(* IEC 61131-3 sources: cc_kush_rewrite/POUs/Dumper/POU/Hardware, 4 files *)

(* ---- FB_DumperConveyorMotors.st ---- *)
FUNCTION_BLOCK FB_DumperConveyorMotors
VAR_INPUT
	Dumper : REFERENCE TO ST_Dumper;
	xStart : BOOL;              // Команда запуска
	xStop : BOOL;               // Команда остановки
	xEmergencyStop : BOOL;      // Аварийная остановка (импульсная)
	xReset : BOOL;              // Сброс аварии (импульсная)
	rTargetFrequency : REAL;    // Целевая частота моторов
END_VAR
VAR_OUTPUT
	eStage : E_StageActuator;   // Текущая стадия
	rCurrentFrequency : REAL;   // Текущая частота моторов (среднее значение)
	xStartingTimeout : BOOL;    // Флаг тайм-аута запуска (STARTING слишком долго)
	xStoppingTimeout : BOOL;    // Флаг тайм-аута остановки (STOPPING слишком долго)
	xVFD_FeedbackLostTimeout : BOOL; // Флаг: потеря обратной связи VFD во время работы (не восстановилась за TIME_TIMEOUT_VFD_FEEDBACK_LOST)
END_VAR
VAR
	STAGE : E_StageActuator := E_StageActuator.IDLE;

	// Подстадии запуска
	nStartingSubstage : INT := 0;
	// 0 - RELEASE_BRAKE: Отпускание тормоза
	// 1 - WAIT_BRAKE_FEEDBACK: Ожидание обратной связи тормоза
	// 2 - START_VFD: Запуск VFD

	// Подстадии остановки
	nStoppingSubstage : INT := 0;
	// 0 - Нормальная работа
	// 1 - STOP_VFD: Остановка VFD
	// 2 - WAIT_VFD_STOP: Ожидание остановки VFD
	// 3 - ACTIVATE_BRAKE: Активация тормоза
	// 4 - WAIT_BRAKE_FEEDBACK: Ожидание обратной связи тормоза

	// Таймер задержки включения тормоза
	tonTimerEnableBrake : TON;

	// Таймер контроля времени запуска (STARTING → WORK)
	tonTimerStarting : TON;

	// Таймер контроля времени остановки (STOPPING → IDLE)
	tonTimerStopping : TON;

	// Таймер контроля потери обратной связи VFD во время работы
	tonTimerVFD_FeedbackLost : TON;

	// Флаг запуска таймера (защита от зацикливания)
	xBrakeTimerStarted : BOOL := FALSE;
END_VAR

// ========================================
// FB_DumperConveyorMotors - Управление моторами конвейера отвалообразователя
// ========================================
//
// НАЗНАЧЕНИЕ:
// - Управление двумя моторами конвейера (22 кВт каждый)
// - Прямой пуск (без плавного разгона)
// - Последовательная остановка (VFD → тормоз)
// - Не знает про ППЗ и верхнеуровневую логику
// - Просто выполняет команды START/STOP
//
// ВХОДЫ:
// - xStart: команда запуска моторов
// - xStop: команда остановки моторов
// - xEmergencyStop: аварийная остановка (импульсная)
// - xReset: сброс аварии (импульсная)
// - rTargetFrequency: целевая частота (Гц)
//
// ВЫХОДЫ:
// - eStage: текущая стадия (IDLE/STARTING/WORK/STOPPING/FAULT)
// - rCurrentFrequency: текущая частота моторов
//
// ========================================

// ========================================
// ПРИОРИТЕТНАЯ ОБРАБОТКА АВАРИЙНОЙ ОСТАНОВКИ
// ========================================

IF xEmergencyStop THEN
	// Аварийная остановка: немедленное выключение VFD
	Dumper.MotorConveyor[1].VFD.qxStart := FALSE;
	Dumper.MotorConveyor[2].VFD.qxStart := FALSE;

	// Активация тормоза
	Dumper.qxBreakerConveyor := FALSE;

	// Переход в FAULT
	STAGE := E_StageActuator.FAULT;
	nStartingSubstage := 0;
	nStoppingSubstage := 0;
	tonTimerEnableBrake(IN := FALSE);
	tonTimerStarting(IN := FALSE);
	tonTimerStopping(IN := FALSE);
	xBrakeTimerStarted := FALSE;
END_IF

// Тайм-аут запуска: если слишком долго в STARTING → аварийная остановка
tonTimerStarting(
	IN := (STAGE = E_StageActuator.STARTING),
	PT := TIME_TIMEOUT_START_DUMPER_CONVEYOR
);

IF tonTimerStarting.Q THEN
	xStartingTimeout := TRUE;
	// Аварийная остановка: немедленное выключение VFD
	Dumper.MotorConveyor[1].VFD.qxStart := FALSE;
	Dumper.MotorConveyor[2].VFD.qxStart := FALSE;
	// Активация тормоза
	Dumper.qxBreakerConveyor := FALSE;
	// Переход в FAULT
	STAGE := E_StageActuator.FAULT;
	nStartingSubstage := 0;
	tonTimerStarting(IN := FALSE);
END_IF

// Тайм-аут остановки: если слишком долго в STOPPING → аварийная остановка
tonTimerStopping(
	IN := (STAGE = E_StageActuator.STOPPING),
	PT := TIME_TIMEOUT_STOP_DUMPER_CONVEYOR
);

IF tonTimerStopping.Q THEN
	xStoppingTimeout := TRUE;
	// Аварийная остановка: немедленное выключение VFD
	Dumper.MotorConveyor[1].VFD.qxStart := FALSE;
	Dumper.MotorConveyor[2].VFD.qxStart := FALSE;
	// Активация тормоза
	Dumper.qxBreakerConveyor := FALSE;
	// Переход в FAULT
	STAGE := E_StageActuator.FAULT;
	nStoppingSubstage := 0;
	tonTimerStopping(IN := FALSE);
END_IF

// Контроль потери обратной связи VFD во время работы
// Если VFD был в работе (WORK) и обратная связь пропала - включаем таймер
// Если обратная связь не вернулась в течение TIME_TIMEOUT_VFD_FEEDBACK_LOST → аварийная остановка
tonTimerVFD_FeedbackLost(
	IN := (STAGE = E_StageActuator.WORK) AND
	      (NOT Dumper.MotorConveyor[1].VFD.fbStateIsWorking.qxSignal
	       OR NOT Dumper.MotorConveyor[2].VFD.fbStateIsWorking.qxSignal),
	PT := TIME_TIMEOUT_VFD_FEEDBACK_LOST
);

IF tonTimerVFD_FeedbackLost.Q THEN
	xVFD_FeedbackLostTimeout := TRUE;
	// Аварийная остановка: немедленное выключение VFD
	Dumper.MotorConveyor[1].VFD.qxStart := FALSE;
	Dumper.MotorConveyor[2].VFD.qxStart := FALSE;
	// Активация тормоза
	Dumper.qxBreakerConveyor := FALSE;
	// Переход в FAULT
	STAGE := E_StageActuator.FAULT;
	tonTimerVFD_FeedbackLost(IN := FALSE);
END_IF

// ========================================
// АВТОМАТ УПРАВЛЕНИЯ МОТОРАМИ
// ========================================

CASE STAGE OF
	E_StageActuator.IDLE:
		// Сброс подстадий
		nStartingSubstage := 0;
		nStoppingSubstage := 0;

		// Сброс флага таймера тормоза
		xBrakeTimerStarted := FALSE;

		// Тормоз активен (удерживает механизм)
		Dumper.qxBreakerConveyor := FALSE;

		// Команда запуска
		IF xStart AND NOT xEmergencyStop THEN
			STAGE := E_StageActuator.STARTING;
		END_IF

	E_StageActuator.STARTING:
		// Проверка команды остановки во время запуска
		IF xStop THEN
			// Прервать запуск и перейти к остановке
			STAGE := E_StageActuator.STOPPING;
			nStartingSubstage := 0;
			nStoppingSubstage := 1; // Начать процедуру остановки
		END_IF

		// Последовательный запуск: Тормоз → VFD → Разгон
		CASE nStartingSubstage OF
			0: // RELEASE_BRAKE - Отпускание тормоза
				// Отпустить тормоз (1 = тормоз отпущен)
				Dumper.qxBreakerConveyor := TRUE;

				// Переход к следующей подстадии
				nStartingSubstage := 1;

			1: // WAIT_BRAKE_FEEDBACK - Ожидание обратной связи тормоза
				// Получить обратную связь реле тормоза
				IF Dumper.fbBreakerConveyor.qxSignal THEN
					// Обратная связь получена, переходим к запуску VFD
					nStartingSubstage := 2;
				END_IF

			2: // START_VFD - Запуск VFD
				// Команда ПУСК на частотный преобразователь
				Dumper.MotorConveyor[1].VFD.qxStart := TRUE;
				Dumper.MotorConveyor[2].VFD.qxStart := TRUE;

				// Если оба VFD запущены (обратная связь)
				IF Dumper.MotorConveyor[1].VFD.fbStateIsWorking.qxSignal
					AND Dumper.MotorConveyor[2].VFD.fbStateIsWorking.qxSignal
				THEN
					// Переход в режим WORK
					STAGE := E_StageActuator.WORK;
					nStartingSubstage := 0;
				END_IF
		END_CASE;

	E_StageActuator.WORK:
		// Нормальная работа
		// Команда остановки - переход в STOPPING
		IF xStop THEN
			STAGE := E_StageActuator.STOPPING;
			nStoppingSubstage := 0;
		END_IF

	E_StageActuator.STOPPING:
		// Штатная остановка через подстадии
		CASE nStoppingSubstage OF
			0: // STOP_VFD - Остановка VFD
				// Отключить команду пуска на VFD
				Dumper.MotorConveyor[1].VFD.qxStart := FALSE;
				Dumper.MotorConveyor[2].VFD.qxStart := FALSE;

				nStoppingSubstage := 1;

			1: // WAIT_VFD_STOP - Ожидание остановки VFD
				// Проверить обратную связь VFD о выключении
				IF NOT Dumper.MotorConveyor[1].VFD.fbStateIsWorking.qxSignal
					AND NOT Dumper.MotorConveyor[2].VFD.fbStateIsWorking.qxSignal
				THEN
					nStoppingSubstage := 2;
				END_IF

			2: // ACTIVATE_BRAKE - Активация тормоза с задержкой
				// Включение таймера на задержку тормоза (один раз)
				IF NOT xBrakeTimerStarted THEN
					xBrakeTimerStarted := TRUE;
				END_IF

				tonTimerEnableBrake(IN := xBrakeTimerStarted, PT := T#5S);

				IF tonTimerEnableBrake.Q THEN
					// Снять сигнал с тормоза (FALSE = активен)
					Dumper.qxBreakerConveyor := FALSE;
					tonTimerEnableBrake(IN := FALSE);
					xBrakeTimerStarted := FALSE;
					nStoppingSubstage := 3;
				END_IF

			3: // Переход в IDLE
				STAGE := E_StageActuator.IDLE;
				nStoppingSubstage := 0;
		END_CASE;

	E_StageActuator.FAULT:
		// Состояние аварии - ожидание сброса
		// Выход из FAULT по команде xReset
		IF xReset THEN
			STAGE := E_StageActuator.IDLE;
			xStartingTimeout := FALSE; // Сброс флага тайм-аута запуска
			xStoppingTimeout := FALSE; // Сброс флага тайм-аута остановки
			xVFD_FeedbackLostTimeout := FALSE; // Сброс флага потери обратной связи VFD
		END_IF
END_CASE;

// ========================================
// ЗАДАНИЕ ЧАСТОТЫ МОТОРОВ
// ========================================

// Установка частоты напрямую в аналоговый выход VFD
// В режимах STARTING и WORK частота = rTargetFrequency (VFD должен знать целевую частоту до запуска)
// В остальных режимах (IDLE, STOPPING, FAULT) частота = 0
IF STAGE = E_StageActuator.STARTING OR STAGE = E_StageActuator.WORK THEN
	Dumper.MotorConveyor[1].VFD.qrOutFrequency := rTargetFrequency;
	Dumper.MotorConveyor[2].VFD.qrOutFrequency := rTargetFrequency;
ELSE
	Dumper.MotorConveyor[1].VFD.qrOutFrequency := 0.0;
	Dumper.MotorConveyor[2].VFD.qrOutFrequency := 0.0;
END_IF;

// ========================================
// ВЫХОДЫ
// ========================================

// Текущая стадия
eStage := STAGE;

// Текущая частота (среднее значение двух моторов)
rCurrentFrequency := (Dumper.MotorConveyor[1].VFD.rActualFrequency
                    + Dumper.MotorConveyor[2].VFD.rActualFrequency) / 2.0;

END_FUNCTION_BLOCK

(* ---- FB_DumperMotorErrors.st ---- *)
FUNCTION_BLOCK FB_DumperMotorErrors
VAR_INPUT
	Dumper : REFERENCE TO ST_Dumper;
	xReset : BOOL; // Команда сброса зафиксированных ошибок
END_VAR
VAR_OUTPUT
	// Ошибки моторов конвейера
	xErrorMotorConv1 : BOOL;
	xErrorMotorConv2 : BOOL;
	xErrorMotorConv_Any : BOOL;

	// Ошибки моторов поворота
	xErrorMotorRot1 : BOOL;
	xErrorMotorRot2 : BOOL;
	xErrorMotorRot_Any : BOOL;

	// Агрегированный выход ошибок
	xErrorMotors : BOOL; // Любая ошибка моторов (VFD failure)

	// Готовность VFD (дискретный сигнал "Готов к пуску")
	xVFD_ReadyConv1 : BOOL; // VFD мотора конвейера 1 готов
	xVFD_ReadyConv2 : BOOL; // VFD мотора конвейера 2 готов
	xVFD_ReadyConv_All : BOOL; // Все VFD конвейера готовы

	xVFD_ReadyRot1 : BOOL; // VFD мотора поворота 1 готов
	xVFD_ReadyRot2 : BOOL; // VFD мотора поворота 2 готов
	xVFD_ReadyRot_All : BOOL; // Все VFD поворота готовы

	xVFD_Ready_All : BOOL; // Все VFD готовы к пуску

	// Состояние автоматических выключателей (QF)
	// TRUE = включен, FALSE = выключен
	// Не является ошибкой, но влияет на готовность к запуску
	xQF_OkConv1 : BOOL; // QF мотора конвейера 1 включен
	xQF_OkConv2 : BOOL; // QF мотора конвейера 2 включен
	xQF_OkConv_All : BOOL; // Все QF конвейера включены

	xQF_OkRot1 : BOOL; // QF мотора поворота 1 включен
	xQF_OkRot2 : BOOL; // QF мотора поворота 2 включен
	xQF_OkRot_All : BOOL; // Все QF поворота включены

	xQF_Ok_All : BOOL; // Все QF включены
END_VAR
VAR
	// Внутренние переменные для текущих состояний ошибок (без фиксации)
	_xCurrentErrorMotorConv1 : BOOL;
	_xCurrentErrorMotorConv2 : BOOL;
	_xCurrentErrorMotorRot1 : BOOL;
	_xCurrentErrorMotorRot2 : BOOL;

	// RS-триггеры для фиксации ошибок
	_fbLatchErrorMotorConv1 : RS;
	_fbLatchErrorMotorConv2 : RS;
	_fbLatchErrorMotorRot1 : RS;
	_fbLatchErrorMotorRot2 : RS;
END_VAR

// ========================================
// FB_DumperMotorErrors - Проверка ошибок моторов отвалообразователя
// ========================================
//
// НАЗНАЧЕНИЕ:
// - Проверка всех моторов отвалообразователя на ошибки
// - Фиксация ошибок через RS-триггеры (память до сброса)
// - Формирование индивидуальных флагов ошибок
// - Агрегирование ошибок
//
// МОТОРЫ:
// - MotorConveyor[1..2]: Моторы конвейера (22 кВт)
// - MotorRotation[1..2]: Моторы поворота (3 кВт)
//
// ПРОВЕРЯЕМЫЕ ОШИБКИ:
// - Ошибка VFD (fbStateFailure: 0 = ошибка, 1 = норма, NC контакт)
//
// ПРОВЕРЯЕМАЯ ГОТОВНОСТЬ:
// - Готовность VFD (fbStateRdyToStart: 1 = готов, 0 = не готов, NO контакт)
//
// ЛОГИКА ФИКСАЦИИ:
// - При возникновении ошибки она фиксируется (SET в RS-триггер)
// - Ошибка сохраняется даже после устранения неисправности
// - Сброс всех зафиксированных ошибок через вход xReset
//
// ========================================

// ========================================
// ПРОВЕРКА МОТОРОВ КОНВЕЙЕРА
// ========================================

// Мотор конвейера 1
// fbStateFailure - NC контакт: 0 = ошибка VFD, 1 = норма
_xCurrentErrorMotorConv1 := NOT Dumper.MotorConveyor[1].VFD.fbStateFailure.qxSignal;

// Мотор конвейера 2
_xCurrentErrorMotorConv2 := NOT Dumper.MotorConveyor[2].VFD.fbStateFailure.qxSignal;

// Фиксируем ошибки через RS-триггеры (SET при ошибке, RESET по команде xReset)
_fbLatchErrorMotorConv1(SET := _xCurrentErrorMotorConv1, RESET1 := xReset);
_fbLatchErrorMotorConv2(SET := _xCurrentErrorMotorConv2, RESET1 := xReset);

// Выходы - зафиксированные ошибки
xErrorMotorConv1 := _fbLatchErrorMotorConv1.Q1;
xErrorMotorConv2 := _fbLatchErrorMotorConv2.Q1;

xErrorMotorConv_Any := xErrorMotorConv1 OR xErrorMotorConv2;

// ========================================
// ПРОВЕРКА МОТОРОВ ПОВОРОТА
// ========================================

// Мотор поворота 1
_xCurrentErrorMotorRot1 := NOT Dumper.MotorRotation[1].VFD.fbStateFailure.qxSignal;

// Мотор поворота 2
_xCurrentErrorMotorRot2 := NOT Dumper.MotorRotation[2].VFD.fbStateFailure.qxSignal;

// Фиксируем ошибки через RS-триггеры (SET при ошибке, RESET по команде xReset)
_fbLatchErrorMotorRot1(SET := _xCurrentErrorMotorRot1, RESET1 := xReset);
_fbLatchErrorMotorRot2(SET := _xCurrentErrorMotorRot2, RESET1 := xReset);

// Выходы - зафиксированные ошибки
xErrorMotorRot1 := _fbLatchErrorMotorRot1.Q1;
xErrorMotorRot2 := _fbLatchErrorMotorRot2.Q1;

xErrorMotorRot_Any := xErrorMotorRot1 OR xErrorMotorRot2;

// ========================================
// АГРЕГИРОВАНИЕ ОШИБОК
// ========================================

xErrorMotors := xErrorMotorConv_Any OR xErrorMotorRot_Any;

// ========================================
// ПРОВЕРКА ГОТОВНОСТИ VFD
// ========================================
// fbStateRdyToStart - NO контакт: 1 = готов к пуску, 0 = не готов
// Готовность проверяется в реальном времени (без фиксации)

// Готовность VFD конвейера
xVFD_ReadyConv1 := Dumper.MotorConveyor[1].VFD.fbStateRdyToStart.qxSignal;
xVFD_ReadyConv2 := Dumper.MotorConveyor[2].VFD.fbStateRdyToStart.qxSignal;
xVFD_ReadyConv_All := xVFD_ReadyConv1 AND xVFD_ReadyConv2;

// Готовность VFD поворота
xVFD_ReadyRot1 := Dumper.MotorRotation[1].VFD.fbStateRdyToStart.qxSignal;
xVFD_ReadyRot2 := Dumper.MotorRotation[2].VFD.fbStateRdyToStart.qxSignal;
xVFD_ReadyRot_All := xVFD_ReadyRot1 AND xVFD_ReadyRot2;

// Общая готовность всех VFD
xVFD_Ready_All := xVFD_ReadyConv_All AND xVFD_ReadyRot_All;

// ========================================
// ПРОВЕРКА СОСТОЯНИЯ АВТОМАТИЧЕСКИХ ВЫКЛЮЧАТЕЛЕЙ (QF)
// ========================================
// fbStateQF - NO контакт: 1 = QF включен, 0 = QF выключен
// Состояние проверяется в реальном времени (без фиксации)
// Выключенный QF - не ошибка, но запуск мотора невозможен

// Состояние QF конвейера
xQF_OkConv1 := Dumper.MotorConveyor[1].fbStateQF.qxSignal;
xQF_OkConv2 := Dumper.MotorConveyor[2].fbStateQF.qxSignal;
xQF_OkConv_All := xQF_OkConv1 AND xQF_OkConv2;

// Состояние QF поворота
xQF_OkRot1 := Dumper.MotorRotation[1].fbStateQF.qxSignal;
xQF_OkRot2 := Dumper.MotorRotation[2].fbStateQF.qxSignal;
xQF_OkRot_All := xQF_OkRot1 AND xQF_OkRot2;

// Общее состояние всех QF
xQF_Ok_All := xQF_OkConv_All AND xQF_OkRot_All;

END_FUNCTION_BLOCK

(* ---- FB_DumperRotationMotors.st ---- *)
FUNCTION_BLOCK FB_DumperRotationMotors
VAR_INPUT
	Dumper : REFERENCE TO ST_Dumper;
	xTurnLeft : BOOL;           // Команда поворота влево
	xTurnRight : BOOL;          // Команда поворота вправо
	xStop : BOOL;               // Команда остановки поворота
	xEmergencyStop : BOOL;      // Аварийная остановка (импульсная)
	xReset : BOOL;              // Сброс аварии (импульсная)
	rTargetFrequency : REAL;    // Целевая частота моторов
END_VAR
VAR_OUTPUT
	eStage : E_StageActuator;   // Текущая стадия
	rCurrentFrequency : REAL;   // Текущая частота моторов (среднее значение)
	xRotatingLeft : BOOL;       // Активен поворот влево
	xRotatingRight : BOOL;      // Активен поворот вправо
	xStartingTimeout : BOOL;    // Флаг тайм-аута запуска (STARTING слишком долго)
	xStoppingTimeout : BOOL;    // Флаг тайм-аута остановки (STOPPING слишком долго)
	xEndSwitchLeftReached : BOOL;   // Достигнут левый концевик
	xEndSwitchRightReached : BOOL;  // Достигнут правый концевик
END_VAR
VAR
	STAGE : E_StageActuator := E_StageActuator.IDLE;

	// Направление поворота
	xLeftActive : BOOL := FALSE;  // Поворот влево активен
	xRightActive : BOOL := FALSE; // Поворот вправо активен

	// Подстадии запуска
	nStartingSubstage : INT := 0;
	// 0 - IDLE
	// 1 - RELEASE_BRAKE: Отпускание тормоза поворота
	// 2 - WAIT_BRAKE_FEEDBACK: Ожидание обратной связи тормоза
	// 3 - START_VFD: Запуск VFD поворота

	// Подстадии остановки
	nStoppingSubstage : INT := 0;
	// 0 - Нормальная работа
	// 1 - STOP_VFD: Остановка VFD
	// 2 - WAIT_VFD_STOP: Ожидание остановки VFD
	// 3 - ACTIVATE_BRAKE: Активация тормоза

	// Таймер задержки включения тормоза
	tonTimerEnableBrake : TON;

	// Таймер контроля времени запуска (STARTING → WORK)
	tonTimerStarting : TON;

	// Таймер контроля времени остановки (STOPPING → IDLE)
	tonTimerStopping : TON;

	// Флаг запуска таймера (защита от зацикливания)
	xBrakeTimerStarted : BOOL := FALSE;
END_VAR

// ========================================
// FB_DumperRotationMotors - Управление моторами поворота отвалообразователя
// ========================================
//
// НАЗНАЧЕНИЕ:
// - Управление двумя моторами поворота (3 кВт каждый)
// - Поддержка реверса (влево/вправо)
// - Блокировка по концевым выключателям
// - Последовательная остановка (VFD → тормоз)
// - Не знает про верхнеуровневую логику
// - Просто выполняет команды TURN_LEFT/TURN_RIGHT/STOP
//
// ВХОДЫ:
// - xTurnLeft: команда поворота влево
// - xTurnRight: команда поворота вправо
// - xStop: команда остановки
// - xEmergencyStop: аварийная остановка (импульсная)
// - xReset: сброс аварии (импульсная)
// - rTargetFrequency: целевая частота (Гц)
//
// ВЫХОДЫ:
// - eStage: текущая стадия (IDLE/STARTING/WORK/STOPPING/FAULT)
// - rCurrentFrequency: текущая частота моторов
// - xRotatingLeft: флаг активного поворота влево
// - xRotatingRight: флаг активного поворота вправо
//
// ========================================

// ========================================
// ПРИОРИТЕТНАЯ ОБРАБОТКА АВАРИЙНОЙ ОСТАНОВКИ
// ========================================

IF xEmergencyStop THEN
	// Аварийная остановка: немедленное выключение VFD
	Dumper.MotorRotation[1].VFD.qxStart := FALSE;
	Dumper.MotorRotation[2].VFD.qxStart := FALSE;
	Dumper.MotorRotation[1].qxVFDReverseStart := FALSE;
	Dumper.MotorRotation[2].qxVFDReverseStart := FALSE;

	// Активация тормоза
	Dumper.qxBreakerRotation := FALSE;

	// Сброс направления
	xLeftActive := FALSE;
	xRightActive := FALSE;

	// Переход в FAULT
	STAGE := E_StageActuator.FAULT;
	nStartingSubstage := 0;
	nStoppingSubstage := 0;
	tonTimerEnableBrake(IN := FALSE);
	tonTimerStarting(IN := FALSE);
	tonTimerStopping(IN := FALSE);
	xBrakeTimerStarted := FALSE;
END_IF

// Тайм-аут запуска: если слишком долго в STARTING → аварийная остановка
tonTimerStarting(
	IN := (STAGE = E_StageActuator.STARTING),
	PT := TIME_TIMEOUT_START_DUMPER_ROTATION
);

IF tonTimerStarting.Q THEN
	xStartingTimeout := TRUE;
	// Аварийная остановка: немедленное выключение VFD
	Dumper.MotorRotation[1].VFD.qxStart := FALSE;
	Dumper.MotorRotation[2].VFD.qxStart := FALSE;
	Dumper.MotorRotation[1].qxVFDReverseStart := FALSE;
	Dumper.MotorRotation[2].qxVFDReverseStart := FALSE;
	// Активация тормоза
	Dumper.qxBreakerRotation := FALSE;
	// Сброс направления
	xLeftActive := FALSE;
	xRightActive := FALSE;
	// Переход в FAULT
	STAGE := E_StageActuator.FAULT;
	nStartingSubstage := 0;
	tonTimerStarting(IN := FALSE);
END_IF

// Тайм-аут остановки: если слишком долго в STOPPING → аварийная остановка
tonTimerStopping(
	IN := (STAGE = E_StageActuator.STOPPING),
	PT := TIME_TIMEOUT_STOP_DUMPER_ROTATION
);

IF tonTimerStopping.Q THEN
	xStoppingTimeout := TRUE;
	// Аварийная остановка: немедленное выключение VFD
	Dumper.MotorRotation[1].VFD.qxStart := FALSE;
	Dumper.MotorRotation[2].VFD.qxStart := FALSE;
	Dumper.MotorRotation[1].qxVFDReverseStart := FALSE;
	Dumper.MotorRotation[2].qxVFDReverseStart := FALSE;
	// Активация тормоза
	Dumper.qxBreakerRotation := FALSE;
	// Сброс направления
	xLeftActive := FALSE;
	xRightActive := FALSE;
	// Переход в FAULT
	STAGE := E_StageActuator.FAULT;
	nStoppingSubstage := 0;
	tonTimerStopping(IN := FALSE);
END_IF

// ========================================
// АВТОМАТ УПРАВЛЕНИЯ МОТОРАМИ ПОВОРОТА
// ========================================

CASE STAGE OF
	E_StageActuator.IDLE:
		// Сброс подстадий
		nStartingSubstage := 0;
		nStoppingSubstage := 0;

		// Сброс флага таймера тормоза
		xBrakeTimerStarted := FALSE;

		// Тормоз активен
		Dumper.qxBreakerRotation := FALSE;

		// Остановка VFD
		Dumper.MotorRotation[1].VFD.qxStart := FALSE;
		Dumper.MotorRotation[2].VFD.qxStart := FALSE;
		Dumper.MotorRotation[1].qxVFDReverseStart := FALSE;
		Dumper.MotorRotation[2].qxVFDReverseStart := FALSE;

		// Сброс флагов направления
		xLeftActive := FALSE;
		xRightActive := FALSE;

		// Команда поворота влево
		IF xTurnLeft AND NOT xEmergencyStop AND NOT xTurnRight THEN
			// Проверка концевого выключателя влево
			// qxSignal = TRUE означает концевик в норме (не нажат)
			IF Dumper.fbEndSwitchLeft.qxSignal THEN
				xLeftActive := TRUE;
				xRightActive := FALSE;
				STAGE := E_StageActuator.STARTING;
			END_IF
		END_IF

		// Команда поворота вправо
		IF xTurnRight AND NOT xEmergencyStop AND NOT xTurnLeft THEN
			// Проверка концевого выключателя вправо
			IF Dumper.fbEndSwitchRight.qxSignal THEN
				xRightActive := TRUE;
				xLeftActive := FALSE;
				STAGE := E_StageActuator.STARTING;
			END_IF
		END_IF

	E_StageActuator.STARTING:
		// Проверка команды остановки во время запуска
		IF xStop THEN
			// Прервать запуск и перейти к остановке
			STAGE := E_StageActuator.STOPPING;
			nStartingSubstage := 0;
			nStoppingSubstage := 0;
		END_IF

		// Проверка достижения концевого выключателя
		IF (xLeftActive AND NOT Dumper.fbEndSwitchLeft.qxSignal)
			OR (xRightActive AND NOT Dumper.fbEndSwitchRight.qxSignal)
		THEN
			// Концевик достигнут, начать остановку
			STAGE := E_StageActuator.STOPPING;
			nStartingSubstage := 0;
			nStoppingSubstage := 0;
		END_IF

		// Последовательный запуск: Тормоз → VFD → Разгон
		CASE nStartingSubstage OF
			0: // IDLE
				nStartingSubstage := 1;

			1: // RELEASE_BRAKE - Отпускание тормоза
				// Отпустить тормоз (1 = тормоз отпущен)
				Dumper.qxBreakerRotation := TRUE;

				// Переход к следующей подстадии
				nStartingSubstage := 2;

			2: // WAIT_BRAKE_FEEDBACK - Ожидание обратной связи тормоза
				// Получить обратную связь реле тормоза
				IF Dumper.fbBreakerRotation.qxSignal THEN
					// Обратная связь получена, переходим к запуску VFD
					nStartingSubstage := 3;
				END_IF

			3: // START_VFD - Запуск VFD
				// Установка направления и запуск VFD
				IF xLeftActive THEN
					// Поворот влево - прямое направление
					Dumper.MotorRotation[1].qxVFDReverseStart := FALSE;
					Dumper.MotorRotation[2].qxVFDReverseStart := FALSE;
					Dumper.MotorRotation[1].VFD.qxStart := TRUE;
					Dumper.MotorRotation[2].VFD.qxStart := TRUE;
				ELSIF xRightActive THEN
					// Поворот вправо - реверс
					Dumper.MotorRotation[1].VFD.qxStart := FALSE;
					Dumper.MotorRotation[2].VFD.qxStart := FALSE;
					Dumper.MotorRotation[1].qxVFDReverseStart := TRUE;
					Dumper.MotorRotation[2].qxVFDReverseStart := TRUE;
				END_IF

				// Проверка запуска VFD (обратная связь)
				IF Dumper.MotorRotation[1].VFD.fbStateIsWorking.qxSignal
					AND Dumper.MotorRotation[2].VFD.fbStateIsWorking.qxSignal
				THEN
					// VFD запущены, переходим в режим работы
					STAGE := E_StageActuator.WORK;
					nStartingSubstage := 0;
				END_IF
		END_CASE;

	E_StageActuator.WORK:
		// Нормальная работа
		// Проверка команды остановки
		IF xStop THEN
			STAGE := E_StageActuator.STOPPING;
			nStoppingSubstage := 0;
		END_IF

		// Проверка достижения концевого выключателя
		IF (xLeftActive AND NOT Dumper.fbEndSwitchLeft.qxSignal)
			OR (xRightActive AND NOT Dumper.fbEndSwitchRight.qxSignal)
		THEN
			// Концевик достигнут, автоматическая остановка
			STAGE := E_StageActuator.STOPPING;
			nStoppingSubstage := 0;
		END_IF

	E_StageActuator.STOPPING:
		// Штатная остановка через подстадии
		CASE nStoppingSubstage OF
			0: // STOP_VFD - Остановка VFD
				// Отключить команду пуска на VFD
				Dumper.MotorRotation[1].VFD.qxStart := FALSE;
				Dumper.MotorRotation[2].VFD.qxStart := FALSE;
				Dumper.MotorRotation[1].qxVFDReverseStart := FALSE;
				Dumper.MotorRotation[2].qxVFDReverseStart := FALSE;

				nStoppingSubstage := 1;

			1: // WAIT_VFD_STOP - Ожидание остановки VFD
				// Проверить обратную связь VFD о выключении
				IF NOT Dumper.MotorRotation[1].VFD.fbStateIsWorking.qxSignal
					AND NOT Dumper.MotorRotation[2].VFD.fbStateIsWorking.qxSignal
				THEN
					nStoppingSubstage := 2;
				END_IF

			2: // ACTIVATE_BRAKE - Активация тормоза с задержкой
				// Включение таймера на задержку тормоза (один раз)
				IF NOT xBrakeTimerStarted THEN
					xBrakeTimerStarted := TRUE;
				END_IF

				tonTimerEnableBrake(IN := xBrakeTimerStarted, PT := T#3S);

				IF tonTimerEnableBrake.Q THEN
					// Снять сигнал с тормоза (FALSE = активен)
					Dumper.qxBreakerRotation := FALSE;
					tonTimerEnableBrake(IN := FALSE);
					xBrakeTimerStarted := FALSE;

					// Сброс флагов направления
					xLeftActive := FALSE;
					xRightActive := FALSE;

					// Переход в IDLE
					STAGE := E_StageActuator.IDLE;
					nStoppingSubstage := 0;
				END_IF
		END_CASE;

	E_StageActuator.FAULT:
		// Состояние аварии - ожидание сброса
		// Выход из FAULT по команде xReset
		IF xReset THEN
			STAGE := E_StageActuator.IDLE;
			xStartingTimeout := FALSE; // Сброс флага тайм-аута запуска
			xStoppingTimeout := FALSE; // Сброс флага тайм-аута остановки
		END_IF
END_CASE;

// ========================================
// ЗАДАНИЕ ЧАСТОТЫ МОТОРОВ
// ========================================

// Установка частоты напрямую в аналоговый выход VFD
// В режимах STARTING и WORK частота = rTargetFrequency (VFD должен знать целевую частоту до запуска)
// В остальных режимах (IDLE, STOPPING, FAULT) частота = 0
IF STAGE = E_StageActuator.STARTING OR STAGE = E_StageActuator.WORK THEN
	Dumper.MotorRotation[1].VFD.qrOutFrequency := rTargetFrequency;
	Dumper.MotorRotation[2].VFD.qrOutFrequency := rTargetFrequency;
ELSE
	Dumper.MotorRotation[1].VFD.qrOutFrequency := 0.0;
	Dumper.MotorRotation[2].VFD.qrOutFrequency := 0.0;
END_IF;

// ========================================
// ВЫХОДЫ
// ========================================

// Текущая стадия
eStage := STAGE;

// Текущая частота (среднее значение двух моторов)
rCurrentFrequency := (Dumper.MotorRotation[1].VFD.rActualFrequency
                    + Dumper.MotorRotation[2].VFD.rActualFrequency) / 2.0;

// Флаги активного поворота
xRotatingLeft := xLeftActive;
xRotatingRight := xRightActive;

// Состояние концевых выключателей (TRUE = концевик достигнут)
// qxSignal = TRUE означает концевик в норме (не нажат), поэтому инвертируем
xEndSwitchLeftReached := NOT Dumper.fbEndSwitchLeft.qxSignal;
xEndSwitchRightReached := NOT Dumper.fbEndSwitchRight.qxSignal;

END_FUNCTION_BLOCK

(* ---- FB_DumperSensors.st ---- *)
FUNCTION_BLOCK FB_DumperSensors
VAR_INPUT
	Dumper : REFERENCE TO ST_Dumper;
	xReset : BOOL; // Команда сброса зафиксированных ошибок

	// Уставки задержки срабатывания для каждого типа датчика
	itDelayZQ_Alarm : TIME;   // Задержка срабатывания датчика схода ленты (Alarm)
	itDelayZQ_Warning : TIME; // Задержка срабатывания датчика схода ленты (Warning)
	itDelayHQ : TIME;         // Задержка срабатывания кабель-тросового выключателя
	itDelaySQ : TIME;         // Задержка срабатывания датчика ограждения барабана
	itDelayGS : TIME;         // Задержка срабатывания датчика заштыбовки
	itDelayYS : TIME;         // Задержка срабатывания датчика продольного разрыва
	itDelayQR : TIME;         // Задержка срабатывания датчика скорости
END_VAR
VAR_OUTPUT
	// Ошибки по датчикам схода ленты (ZQ Alarm)
	xErrorZQ1 : BOOL;
	xErrorZQ2 : BOOL;
	xErrorZQ3 : BOOL;
	xErrorZQ4 : BOOL;
	xErrorZQ_Any : BOOL; // Любая ошибка ZQ

	// Предупреждения по датчикам схода ленты (ZQ Warning)
	xWarningZQ1 : BOOL;
	xWarningZQ2 : BOOL;
	xWarningZQ3 : BOOL;
	xWarningZQ4 : BOOL;
	xWarningZQ_Any : BOOL; // Любое предупреждение ZQ

	// Ошибки по кабель-тросовым выключателям (HQ)
	xErrorHQ1 : BOOL;
	xErrorHQ2 : BOOL;
	xErrorHQ3 : BOOL;
	xErrorHQ4 : BOOL;
	xErrorHQ_Any : BOOL; // Любая ошибка HQ

	// Ошибки по ограждениям барабана (SQ)
	xErrorSQ1 : BOOL;
	xErrorSQ2 : BOOL;
	xErrorSQ_Any : BOOL; // Любая ошибка SQ

	// Ошибка контроля заштыбовки (GS)
	xErrorGS : BOOL;

	// Ошибки датчиков скорости (QR)
	xErrorQR1 : BOOL;
	xErrorQR2 : BOOL;
	xErrorQR_Any : BOOL; // Любая ошибка QR

	// Ошибка контроля продольного разрыва (YS)
	xErrorYS : BOOL;

	// Агрегированные выходы
	xErrorSafetySensors : BOOL;  // Любая ошибка датчиков безопасности
	xWarningSafetySensors : BOOL; // Любое предупреждение датчиков безопасности
END_VAR
VAR
	// Внутренние переменные для фиксации ошибок (текущие состояния без фиксации)
	_xCurrentErrorZQ1 : BOOL;
	_xCurrentErrorZQ2 : BOOL;
	_xCurrentErrorZQ3 : BOOL;
	_xCurrentErrorZQ4 : BOOL;

	_xCurrentWarningZQ1 : BOOL;
	_xCurrentWarningZQ2 : BOOL;
	_xCurrentWarningZQ3 : BOOL;
	_xCurrentWarningZQ4 : BOOL;

	_xCurrentErrorHQ1 : BOOL;
	_xCurrentErrorHQ2 : BOOL;
	_xCurrentErrorHQ3 : BOOL;
	_xCurrentErrorHQ4 : BOOL;

	_xCurrentErrorSQ1 : BOOL;
	_xCurrentErrorSQ2 : BOOL;

	_xCurrentErrorGS : BOOL;
	_xCurrentErrorQR1 : BOOL;
	_xCurrentErrorQR2 : BOOL;
	_xCurrentErrorYS : BOOL;

	// RS-триггеры для фиксации ошибок
	_fbLatchErrorZQ1 : RS;
	_fbLatchErrorZQ2 : RS;
	_fbLatchErrorZQ3 : RS;
	_fbLatchErrorZQ4 : RS;

	_fbLatchWarningZQ1 : RS;
	_fbLatchWarningZQ2 : RS;
	_fbLatchWarningZQ3 : RS;
	_fbLatchWarningZQ4 : RS;

	_fbLatchErrorHQ1 : RS;
	_fbLatchErrorHQ2 : RS;
	_fbLatchErrorHQ3 : RS;
	_fbLatchErrorHQ4 : RS;

	_fbLatchErrorSQ1 : RS;
	_fbLatchErrorSQ2 : RS;

	_fbLatchErrorGS : RS;
	_fbLatchErrorQR1 : RS;
	_fbLatchErrorQR2 : RS;
	_fbLatchErrorYS : RS;

	// TON таймеры задержки срабатывания для каждого датчика
	// Датчики схода ленты (ZQ Alarm)
	_fbDelayZQ1Alarm : TON;
	_fbDelayZQ2Alarm : TON;
	_fbDelayZQ3Alarm : TON;
	_fbDelayZQ4Alarm : TON;

	// Датчики схода ленты (ZQ Warning)
	_fbDelayZQ1Warning : TON;
	_fbDelayZQ2Warning : TON;
	_fbDelayZQ3Warning : TON;
	_fbDelayZQ4Warning : TON;

	// Кабель-тросовые выключатели (HQ)
	_fbDelayHQ1 : TON;
	_fbDelayHQ2 : TON;
	_fbDelayHQ3 : TON;
	_fbDelayHQ4 : TON;

	// Ограждения барабана (SQ)
	_fbDelaySQ1 : TON;
	_fbDelaySQ2 : TON;

	// Заштыбовка (GS)
	_fbDelayGS : TON;

	// Датчики скорости (QR)
	_fbDelayQR1 : TON;
	_fbDelayQR2 : TON;

	// Продольный разрыв (YS)
	_fbDelayYS : TON;
END_VAR

// ========================================
// FB_DumperSensors - Обработка датчиков безопасности отвалообразователя
// ========================================
//
// НАЗНАЧЕНИЕ:
// - Мониторинг всех датчиков безопасности
// - Фиксация ошибок через RS-триггеры (память до сброса)
// - Формирование индивидуальных флагов ошибок
// - Агрегирование ошибок и предупреждений
//
// ДАТЧИКИ:
// - ZQ (1-4): Контроль схода ленты (Alarm + Warning)
// - HQ (1-4): Кабель-тросовый выключатель (аварийная остановка)
// - SQ (1-2): Контроль ограждения барабана
// - GS: Контроль заштыбовки
// - QR (1-2): Измерение скорости вращения барабана
// - YS: Контроль продольного разрыва ленты
//
// ЛОГИКА ФИКСАЦИИ:
// - При возникновении ошибки она фиксируется (SET в RS-триггер)
// - Ошибка сохраняется даже после устранения неисправности датчика
// - Сброс всех зафиксированных ошибок через вход xReset
//
// ВЫХОДЫ:
// - Индивидуальные флаги для каждого датчика (зафиксированные)
// - Агрегированные флаги (Any) для групп датчиков
// - Общие флаги ошибок и предупреждений
//
// ========================================

// ========================================
// ДАТЧИКИ СХОДА ЛЕНТЫ (ZQ) - ALARM
// ========================================
// Логика: 1 = Норма, 0 = Тревога (сход ленты)

// Таймеры задержки срабатывания (сигнал должен удерживаться itDelayZQ_Alarm перед фиксацией)
_fbDelayZQ1Alarm(IN := NOT Dumper.fbZQAlarm[1].qxSignal, PT := itDelayZQ_Alarm);
_fbDelayZQ2Alarm(IN := NOT Dumper.fbZQAlarm[2].qxSignal, PT := itDelayZQ_Alarm);
_fbDelayZQ3Alarm(IN := NOT Dumper.fbZQAlarm[3].qxSignal, PT := itDelayZQ_Alarm);
_fbDelayZQ4Alarm(IN := NOT Dumper.fbZQAlarm[4].qxSignal, PT := itDelayZQ_Alarm);

// Определяем текущее состояние датчиков (после задержки)
_xCurrentErrorZQ1 := _fbDelayZQ1Alarm.Q;
_xCurrentErrorZQ2 := _fbDelayZQ2Alarm.Q;
_xCurrentErrorZQ3 := _fbDelayZQ3Alarm.Q;
_xCurrentErrorZQ4 := _fbDelayZQ4Alarm.Q;

// Фиксируем ошибки через RS-триггеры (SET при ошибке, RESET по команде xReset)
_fbLatchErrorZQ1(SET := _xCurrentErrorZQ1, RESET1 := xReset);
_fbLatchErrorZQ2(SET := _xCurrentErrorZQ2, RESET1 := xReset);
_fbLatchErrorZQ3(SET := _xCurrentErrorZQ3, RESET1 := xReset);
_fbLatchErrorZQ4(SET := _xCurrentErrorZQ4, RESET1 := xReset);

// Выходы - зафиксированные ошибки
xErrorZQ1 := _fbLatchErrorZQ1.Q1;
xErrorZQ2 := _fbLatchErrorZQ2.Q1;
xErrorZQ3 := _fbLatchErrorZQ3.Q1;
xErrorZQ4 := _fbLatchErrorZQ4.Q1;

xErrorZQ_Any := xErrorZQ1 OR xErrorZQ2 OR xErrorZQ3 OR xErrorZQ4;

// ========================================
// ДАТЧИКИ СХОДА ЛЕНТЫ (ZQ) - WARNING
// ========================================
// Логика: 1 = Норма, 0 = Предупреждение (лента близка к сходу)

// Таймеры задержки срабатывания (сигнал должен удерживаться itDelayZQ_Warning перед фиксацией)
_fbDelayZQ1Warning(IN := NOT Dumper.fbZQWarning[1].qxSignal, PT := itDelayZQ_Warning);
_fbDelayZQ2Warning(IN := NOT Dumper.fbZQWarning[2].qxSignal, PT := itDelayZQ_Warning);
_fbDelayZQ3Warning(IN := NOT Dumper.fbZQWarning[3].qxSignal, PT := itDelayZQ_Warning);
_fbDelayZQ4Warning(IN := NOT Dumper.fbZQWarning[4].qxSignal, PT := itDelayZQ_Warning);

// Определяем текущее состояние датчиков (после задержки)
_xCurrentWarningZQ1 := _fbDelayZQ1Warning.Q;
_xCurrentWarningZQ2 := _fbDelayZQ2Warning.Q;
_xCurrentWarningZQ3 := _fbDelayZQ3Warning.Q;
_xCurrentWarningZQ4 := _fbDelayZQ4Warning.Q;

// Фиксируем предупреждения через RS-триггеры
_fbLatchWarningZQ1(SET := _xCurrentWarningZQ1, RESET1 := xReset);
_fbLatchWarningZQ2(SET := _xCurrentWarningZQ2, RESET1 := xReset);
_fbLatchWarningZQ3(SET := _xCurrentWarningZQ3, RESET1 := xReset);
_fbLatchWarningZQ4(SET := _xCurrentWarningZQ4, RESET1 := xReset);

// Выходы - зафиксированные предупреждения
xWarningZQ1 := _fbLatchWarningZQ1.Q1;
xWarningZQ2 := _fbLatchWarningZQ2.Q1;
xWarningZQ3 := _fbLatchWarningZQ3.Q1;
xWarningZQ4 := _fbLatchWarningZQ4.Q1;

xWarningZQ_Any := xWarningZQ1 OR xWarningZQ2 OR xWarningZQ3 OR xWarningZQ4;

// ========================================
// КАБЕЛЬ-ТРОСОВЫЕ ВЫКЛЮЧАТЕЛИ (HQ)
// ========================================
// Логика: 1 = Норма, 0 = Аварийная остановка (трос натянут)

// Таймеры задержки срабатывания (сигнал должен удерживаться itDelayHQ перед фиксацией)
_fbDelayHQ1(IN := NOT Dumper.fbHQ_IsOk[1].qxSignal, PT := itDelayHQ);
_fbDelayHQ2(IN := NOT Dumper.fbHQ_IsOk[2].qxSignal, PT := itDelayHQ);
_fbDelayHQ3(IN := NOT Dumper.fbHQ_IsOk[3].qxSignal, PT := itDelayHQ);
_fbDelayHQ4(IN := NOT Dumper.fbHQ_IsOk[4].qxSignal, PT := itDelayHQ);

// Определяем текущее состояние датчиков (после задержки)
_xCurrentErrorHQ1 := _fbDelayHQ1.Q;
_xCurrentErrorHQ2 := _fbDelayHQ2.Q;
_xCurrentErrorHQ3 := _fbDelayHQ3.Q;
_xCurrentErrorHQ4 := _fbDelayHQ4.Q;

// Фиксируем ошибки через RS-триггеры
_fbLatchErrorHQ1(SET := _xCurrentErrorHQ1, RESET1 := xReset);
_fbLatchErrorHQ2(SET := _xCurrentErrorHQ2, RESET1 := xReset);
_fbLatchErrorHQ3(SET := _xCurrentErrorHQ3, RESET1 := xReset);
_fbLatchErrorHQ4(SET := _xCurrentErrorHQ4, RESET1 := xReset);

// Выходы - зафиксированные ошибки
xErrorHQ1 := _fbLatchErrorHQ1.Q1;
xErrorHQ2 := _fbLatchErrorHQ2.Q1;
xErrorHQ3 := _fbLatchErrorHQ3.Q1;
xErrorHQ4 := _fbLatchErrorHQ4.Q1;

xErrorHQ_Any := xErrorHQ1 OR xErrorHQ2 OR xErrorHQ3 OR xErrorHQ4;

// ========================================
// КОНТРОЛЬ ОГРАЖДЕНИЯ БАРАБАНА (SQ)
// ========================================
// Логика: 1 = Норма (ограждение закрыто), 0 = Тревога (ограждение открыто)

// Таймеры задержки срабатывания (сигнал должен удерживаться itDelaySQ перед фиксацией)
_fbDelaySQ1(IN := NOT Dumper.fbSQ_IsOk[1].qxSignal, PT := itDelaySQ);
_fbDelaySQ2(IN := NOT Dumper.fbSQ_IsOk[2].qxSignal, PT := itDelaySQ);

// Определяем текущее состояние датчиков (после задержки)
_xCurrentErrorSQ1 := _fbDelaySQ1.Q;
_xCurrentErrorSQ2 := _fbDelaySQ2.Q;

// Фиксируем ошибки через RS-триггеры
_fbLatchErrorSQ1(SET := _xCurrentErrorSQ1, RESET1 := xReset);
_fbLatchErrorSQ2(SET := _xCurrentErrorSQ2, RESET1 := xReset);

// Выходы - зафиксированные ошибки
xErrorSQ1 := _fbLatchErrorSQ1.Q1;
xErrorSQ2 := _fbLatchErrorSQ2.Q1;

xErrorSQ_Any := xErrorSQ1 OR xErrorSQ2;

// ========================================
// КОНТРОЛЬ ЗАШТЫБОВКИ (GS)
// ========================================
// Логика: 1 = Норма, 0 = Тревога (заштыбовка материала)

// Таймер задержки срабатывания (сигнал должен удерживаться itDelayGS перед фиксацией)
_fbDelayGS(IN := NOT Dumper.fbGS1.qxSignal, PT := itDelayGS);

// Определяем текущее состояние датчика (после задержки)
_xCurrentErrorGS := _fbDelayGS.Q;

// Фиксируем ошибку через RS-триггер
_fbLatchErrorGS(SET := _xCurrentErrorGS, RESET1 := xReset);

// Выход - зафиксированная ошибка
xErrorGS := _fbLatchErrorGS.Q1;

// ========================================
// ДАТЧИКИ СКОРОСТИ (QR)
// ========================================
// Логика: Проверка наличия импульсов (детектирование остановки при работающем моторе)
// Ошибка определяется на верхнем уровне по сравнению с состоянием мотора

// Таймеры задержки срабатывания (резерв для будущей реализации)
_fbDelayQR1(IN := FALSE, PT := itDelayQR); // Резерв для будущей реализации
_fbDelayQR2(IN := FALSE, PT := itDelayQR); // Резерв для будущей реализации

// Определяем текущее состояние датчиков (после задержки)
_xCurrentErrorQR1 := _fbDelayQR1.Q;
_xCurrentErrorQR2 := _fbDelayQR2.Q;

// Фиксируем ошибки через RS-триггеры
_fbLatchErrorQR1(SET := _xCurrentErrorQR1, RESET1 := xReset);
_fbLatchErrorQR2(SET := _xCurrentErrorQR2, RESET1 := xReset);

// Выходы - зафиксированные ошибки
xErrorQR1 := _fbLatchErrorQR1.Q1;
xErrorQR2 := _fbLatchErrorQR2.Q1;

xErrorQR_Any := xErrorQR1 OR xErrorQR2;

// ========================================
// КОНТРОЛЬ ПРОДОЛЬНОГО РАЗРЫВА (YS)
// ========================================
// Логика: 1 = Норма, 0 = Тревога (продольный разрыв ленты)

// Таймер задержки срабатывания (сигнал должен удерживаться itDelayYS перед фиксацией)
_fbDelayYS(IN := NOT Dumper.fbYS1.qxSignal, PT := itDelayYS);

// Определяем текущее состояние датчика (после задержки)
_xCurrentErrorYS := _fbDelayYS.Q;

// Фиксируем ошибку через RS-триггер
_fbLatchErrorYS(SET := _xCurrentErrorYS, RESET1 := xReset);

// Выход - зафиксированная ошибка
xErrorYS := _fbLatchErrorYS.Q1;

// ========================================
// АГРЕГИРОВАНИЕ ОШИБОК И ПРЕДУПРЕЖДЕНИЙ
// ========================================

// Все критические ошибки датчиков безопасности
xErrorSafetySensors := xErrorZQ_Any    // Сход ленты (критический уровень)
                    OR xErrorHQ_Any     // Аварийная остановка по тросу
                    OR xErrorSQ_Any     // Открыто ограждение
                    OR xErrorGS         // Заштыбовка
                    OR xErrorQR_Any     // Остановка барабана
                    OR xErrorYS;        // Продольный разрыв

// Все предупреждения датчиков безопасности
xWarningSafetySensors := xWarningZQ_Any; // Предупреждение схода ленты

END_FUNCTION_BLOCK
